(* IEC 61131-3 sources: RL_MAR/experiments/comparison/autoplc/results/deepseek-ai-DeepSeek-V3.2_20260508_111905/med_82, 1 file *)

(* ---- med_82_1.st ---- *)
FUNCTION_BLOCK PetFeederControl
VAR_INPUT
    CurrentTime : TIME; (* Current system time input *)
END_VAR
VAR_OUTPUT
    FoodDispense : BOOL; (* Food dispenser control signal *)
END_VAR
VAR
    FeedTime1 : TIME := T#8H0M0S; (* First feeding time - 8:00 AM *)
    FeedTime2 : TIME := T#12H0M0S; (* Second feeding time - 12:00 PM *)
    FeedTime3 : TIME := T#18H0M0S; (* Third feeding time - 6:00 PM *)
    FoodAmount : INT := 50; (* Amount of food to dispense in grams *)
END_VAR

    (* Main control logic *)
    FoodDispense := FALSE;

    (* Check if current time is within first feeding window *)
    IF (CurrentTime >= FeedTime1) AND (CurrentTime < (FeedTime1 + T#30S)) THEN
        FoodDispense := TRUE;
    END_IF;

    (* Check if current time is within second feeding window *)
    IF (CurrentTime >= FeedTime2) AND (CurrentTime < (FeedTime2 + T#30S)) THEN
        FoodDispense := TRUE;
    END_IF;

    (* Check if current time is within third feeding window *)
    IF (CurrentTime >= FeedTime3) AND (CurrentTime < (FeedTime3 + T#30S)) THEN
        FoodDispense := TRUE;
    END_IF;

END_FUNCTION_BLOCK
